# EPICS substitutions: support/ebrick/2-2-3/iocBoot/iocebrick/ebrickPOSDAC.substitutions
file ../../db/ebrDAC.db
{
pattern
{P         H       F       D       PREC    CH  MIN     MAX     PORT }

{ebrick:   pos01:  ana01:  ao01    3       0   -10     10      POSDAC }
{ebrick:   pos01:  ana01:  ao02    3       1   -10     10      POSDAC }
{ebrick:   pos01:  ana01:  ao03    3       2   -10     10      POSDAC }
{ebrick:   pos01:  ana01:  ao04    3       3   -10     10      POSDAC }

}
